NETWORK
TITLE = S006::STEP 006:TRAN 007: Pressure below setpoint?
//----------------------------------------------------------------------------//
// TRAN   TRAN   TRAN   TRAN   TRAN   TRAN   TRAN   TRAN   TRAN   TRAN   TRAN //
// TRAN   TRAN   TRAN   TRAN   TRAN   TRAN   TRAN   TRAN   TRAN   TRAN   TRAN //
//----------------------------------------------------------------------------//
// Pressure reduced below PRES_VAC.
//----------------------------------------------------------------------------//
// CONDITION   CONDITION   CONDITION   CONDITION   CONDITION   CONDITION   CO //
// CONDITION   CONDITION   CONDITION   CONDITION   CONDITION   CONDITION   CO //
//----------------------------------------------------------------------------//
      A(;
      L #_emc_gas_pi_vessel_pv;
      L #_r_pres_vac;
      <R;
      );






  //============================= TRAN FOOTER ==============================//
  // Transition jump control:                                               //
  //------------------------------------------------------------------------//
      A #sqSequencer.STEP.JumpCtrl;
      S #sqSequencer.STEP.Jump;
      S #sqSequencer.STEP.jumpDone[06];

NETWORK
TITLE = S006:t007::TRANS-v: EXIT TRANSITION AND READY THE NEXT STEP
//------------------------------------------------------------------------//
// Check the jump flag and jump to the next step if the transition        //
// condition is true and has set the jump flag:                           //
//------------------------------------------------------------------------//
      A #sqSequencer.STEP.Jump;
      JCN x007;

      R #sqSequencer.STEP.Jump;
      R #sqSequencer.STEP.Finished;

      L 08   ;// Load next STEPNO to jump to if transition satisfied
      T #sqSequencer.STEP.NumberNext;//Next Step08.

      JU COMM            ;// Transition satisfied, Exit, go to next step
x007:      NOP 0;






NETWORK
TITLE = S006::STEP-006:EXIT TRANSITION:
//========================== STEP TRANSFER ===============================//
// Jump to the common step progression code:                              //
//------------------------------------------------------------------------//
      JU COMM;






NETWORK
TITLE = S007: STEP-07::UO_MX_SETUP : Vacuum hold evacuation failed
//================================ STEP HEADER ===========================//
// STEP007 STEP007 STEP007 STEP007
// AUTOCODE   AUTOCODE   AUTOCODE   AUTOCODE   AUTOCODE   AUTOCODE   AUTO //
// STEP007 STEP007 STEP007 STEP007
//------------------------------------------------------------------------//
// Raise vacuum failed message.
// Log vacuum ejector time failed.
// Prompt operator to confirm to try again.
//------------------------------------------------------------------------//
S007:      NOP 0;

      SET;
      R #sqSequencer.STEP.jumpDone[07];
      A #sqSequencer.CMD.Pause;//If paused jump
      JC COMM;

NETWORK
TITLE = S007:STEP-07:Begin Action

      A #sqSequencer.STEP.Finished;
      JC A007;// Exit Action code, Jump to A007 Transition code

    //----------------------------------------------------------------------//
    // Begin step Action:                                                   //
    //----------------------------------------------------------------------//
      A #sqSequencer.STEP.Active;
      JC L007;// Action number loaded, Jump to L007--Step Action List

    //----------------------------------------------------------------------//
    // Load Default/Initial Step action number:                             //
    //----------------------------------------------------------------------//
      S #sqSequencer.STEP.Active;
      S #sqStepTimer.IN;
      L 1;//First Action, Step must contain Minimum one action
      T #sqSequencer.STEP.ActionNumber;

//----------------------------------------------------------------------------//
// Step action list.                                                          //
// aann=mini Action step number(aa) inside main step number(nn)               //
// First Action aa00, Second action ab00, Third ac00, etc.                    //
//----------------------------------------------------------------------------//
L007:      NOP 0;

      L #sqSequencer.STEP.ActionNumber;
      JL r007;//Wrong Action number
      JU _007;//Action error handling
      JU aa07;//ACTION-01


//----------------------------------------------------------------------------//
// More step action in the list can be inserted here, upto ab is tested:      //
//----------------------------------------------------------------------------//
r007:      NOP 0;//Wrong action number
      S #sqSequencer.Error_Fault;
      JU k007;//Exit
_007:      NOP 0;// Action error handling
      JU k007;// Exit






NETWORK
TITLE = S007:: STEP-007:: : ACTION CODE
//================================ ACT HEADER ============================//
// ACTION ACTION ACTION ACTION ACTION ACTION ACTION ACTION ACTION ACTION  //
// AUTOCODE   AUTOCODE   AUTOCODE   AUTOCODE   AUTOCODE   AUTOCODE   AUTO //
// ACTION ACTION ACTION ACTION ACTION ACTION ACTION ACTION ACTION ACTION  //
//------------------------------------------------------------------------//
// //Raise vacuum failed message.
// //Log vacuum time failed.
// //Prompt operator to confirm to try again.
aa07:      NOP 0;

  //------------------------------------------------------------------------//
  // ACT ACT ACT ACT ACT ACT ACT ACT ACT ACT ACT ACT ACT ACT ACT ACT ACT    //
  //------------------------------------------------------------------------//
  //Set flag to raise vacuum failed message
      SET;
      S #_log_real_vacuum_fail;
      S #_prompt_not_reach;

//Log pressure after vacuum timer expired(TIME_EJECT failed).
      L #_emc_gas_pi_vessel_pv;
      T #_real_vacuum_fail;

  //------------------------------------------------------------------------//
  // VERIFY  VERIFY VERIFY VERIFY VERIFY VERIFY VERIFY VERIFY VERIFY VERIFY //
  //------------------------------------------------------------------------//
      A "uncondJump";
      S #sqSequencer.STEP.ActionVerified;//Action verified

  //------------------------------------------------------------------------//
  // Action done:                                                           //
  //------------------------------------------------------------------------//
      O #sqSequencer.STEP.ActionVerified;
      O #smc.NO_VERIFIC     ;//No verification , bypass verification code
      S #sqSequencer.STEP.ActionFinished;






  //============================= STEP FOOTER ==============================//
  // AUTOCODE   AUTOCODE   AUTOCODE   AUTOCODE   AUTOCODE   AUTOCODE   AUTO //
  // Get Ready after action finished:                                       //
  //------------------------------------------------------------------------//
      A #sqSequencer.STEP.ActionFinished;
      JCN k007;

  //------------------------------------------------------------------------//
  // Reset Action finished flag, ready for next step action:                //
  //------------------------------------------------------------------------//
      R #sqSequencer.STEP.ActionVerified;
      R #sqSequencer.STEP.ActionFinished;

  //------------------------------------------------------------------------//
  // If ALL actions are finished:                                           //
  //------------------------------------------------------------------------//
      SET;
      S #sqSequencer.STEP.Finished;
      R #sqSequencer.STEP.Active;
      S #sqSequencer.STEP.Done[07];

  //------------------------------------------------------------------------//
  // End Step action(s):                                                    //
  //------------------------------------------------------------------------//
      JU k007;

//----------------------------------------------------------------------------//
// Finished Step Action(s):                                                   //
//----------------------------------------------------------------------------//
k007:      NOP 0;

      A #sqStepTimerExpired;
      S #sqSequencer.STEP.WithError[07];// Step error flag
      S #sqSequencer.Error_Fault;
      R #sqStepTimer.IN;

NETWORK
TITLE = S007:STEP-007::Begin Transition
//------------------------------------------------------------------------//
// Begin the transition code:                                             //
//------------------------------------------------------------------------//
A007:      NOP 0;
      R #sqStepTimer.IN;






  //============================= TRAN HEADER ==============================//
  // AUTOCODE   AUTOCODE   AUTOCODE   AUTOCODE   AUTOCODE   AUTOCODE   AUTO //
  // Bypass transition if manual jump:                                      //
  //------------------------------------------------------------------------//
      A #sqSequencer.STEP.Finished;
      A #smc.TRN_AND_JUMP   ;//Manual jump is set Transition as bypassed
      JCN COMM            ;//exit

NETWORK
TITLE = S007::STEP 007:TRAN 008: Try again?
//----------------------------------------------------------------------------//
// TRAN   TRAN   TRAN   TRAN   TRAN   TRAN   TRAN   TRAN   TRAN   TRAN   TRAN //
// TRAN   TRAN   TRAN   TRAN   TRAN   TRAN   TRAN   TRAN   TRAN   TRAN   TRAN //
//----------------------------------------------------------------------------//
// Operator want to try again.
//----------------------------------------------------------------------------//
// CONDITION   CONDITION   CONDITION   CONDITION   CONDITION   CONDITION   CO //
// CONDITION   CONDITION   CONDITION   CONDITION   CONDITION   CONDITION   CO //
//----------------------------------------------------------------------------//
      A #_prompt_not_reach_confirm_yes;






  //============================= TRAN FOOTER ==============================//
  // Transition jump control:                                               //
  //------------------------------------------------------------------------//
      A #sqSequencer.STEP.JumpCtrl;
      S #sqSequencer.STEP.Jump;
      S #sqSequencer.STEP.jumpDone[07];

NETWORK
TITLE = S007:t008::TRANS-v: EXIT TRANSITION AND READY THE NEXT STEP
//------------------------------------------------------------------------//
// Check the jump flag and jump to the next step if the transition        //
// condition is true and has set the jump flag:                           //
//------------------------------------------------------------------------//
      A #sqSequencer.STEP.Jump;
      JCN x008;

      R #sqSequencer.STEP.Jump;
      R #sqSequencer.STEP.Finished;

      L 09   ;// Load next STEPNO to jump to if transition satisfied
      T #sqSequencer.STEP.NumberNext;//Next Step09.

      JU COMM            ;// Transition satisfied, Exit, go to next step
x008:      NOP 0;






  //============================= TRAN HEADER ==============================//
  // AUTOCODE   AUTOCODE   AUTOCODE   AUTOCODE   AUTOCODE   AUTOCODE   AUTO //
  // Bypass transition if manual jump:                                      //
  //------------------------------------------------------------------------//
      A #sqSequencer.STEP.Finished;
      A #smc.TRN_AND_JUMP   ;//Manual jump is set Transition as bypassed
      JCN COMM            ;//exit

NETWORK
TITLE = S007::STEP 007:TRAN 009: No try?
//----------------------------------------------------------------------------//
// TRAN   TRAN   TRAN   TRAN   TRAN   TRAN   TRAN   TRAN   TRAN   TRAN   TRAN //
// TRAN   TRAN   TRAN   TRAN   TRAN   TRAN   TRAN   TRAN   TRAN   TRAN   TRAN //
//----------------------------------------------------------------------------//
// Operator don't want to try again.
//----------------------------------------------------------------------------//
// CONDITION   CONDITION   CONDITION   CONDITION   CONDITION   CONDITION   CO //
// CONDITION   CONDITION   CONDITION   CONDITION   CONDITION   CONDITION   CO //
//----------------------------------------------------------------------------//
      A #_prompt_not_reach_confirm_no;






  //============================= TRAN FOOTER ==============================//
  // Transition jump control:                                               //
  //------------------------------------------------------------------------//
      A #sqSequencer.STEP.JumpCtrl;
      S #sqSequencer.STEP.Jump;
      S #sqSequencer.STEP.jumpDone[07];

NETWORK
TITLE = S007:t009::TRANS-v: EXIT TRANSITION AND READY THE NEXT STEP
//------------------------------------------------------------------------//
// Check the jump flag and jump to the next step if the transition        //
// condition is true and has set the jump flag:                           //
//------------------------------------------------------------------------//
      A #sqSequencer.STEP.Jump;
      JCN x009;

      R #sqSequencer.STEP.Jump;
      R #sqSequencer.STEP.Finished;

      L 10   ;// Load next STEPNO to jump to if transition satisfied
      T #sqSequencer.STEP.NumberNext;//Next Step10.

      JU COMM            ;// Transition satisfied, Exit, go to next step
x009:      NOP 0;






NETWORK
TITLE = S007::STEP-007:EXIT TRANSITION:
//========================== STEP TRANSFER ===============================//
// Jump to the common step progression code:                              //
//------------------------------------------------------------------------//
      JU COMM;






NETWORK
TITLE = S008: STEP-08::UO_MX_SETUP : Start Vacuum Hold Timer
//================================ STEP HEADER ===========================//
// STEP008 STEP008 STEP008 STEP008
// AUTOCODE   AUTOCODE   AUTOCODE   AUTOCODE   AUTOCODE   AUTOCODE   AUTO //
// STEP008 STEP008 STEP008 STEP008
//------------------------------------------------------------------------//
// Close Mx vent line vacuum valve.
// Start Vacuum  Hold Timer.
// Store Vacuum Hold test begin time.
//------------------------------------------------------------------------//
S008:      NOP 0;

      SET;
      R #sqSequencer.STEP.jumpDone[08];
      A #sqSequencer.CMD.Pause;//If paused jump
      JC COMM;

NETWORK
TITLE = S008:STEP-08:Begin Action

      A #sqSequencer.STEP.Finished;
      JC A008;// Exit Action code, Jump to A008 Transition code

    //----------------------------------------------------------------------//
    // Begin step Action:                                                   //
    //----------------------------------------------------------------------//
      A #sqSequencer.STEP.Active;
      JC L008;// Action number loaded, Jump to L008--Step Action List

    //----------------------------------------------------------------------//
    // Load Default/Initial Step action number:                             //
    //----------------------------------------------------------------------//
      S #sqSequencer.STEP.Active;
      S #sqStepTimer.IN;
      L 1;//First Action, Step must contain Minimum one action
      T #sqSequencer.STEP.ActionNumber;

//----------------------------------------------------------------------------//
// Step action list.                                                          //
// aann=mini Action step number(aa) inside main step number(nn)               //
// First Action aa00, Second action ab00, Third ac00, etc.                    //
//----------------------------------------------------------------------------//
L008:      NOP 0;

      L #sqSequencer.STEP.ActionNumber;
      JL r008;//Wrong Action number
      JU _008;//Action error handling
      JU aa08;//ACTION-01
      JU ab08;//ACTION-02


//----------------------------------------------------------------------------//
// More step action in the list can be inserted here, upto ab is tested:      //
//----------------------------------------------------------------------------//
r008:      NOP 0;//Wrong action number
      S #sqSequencer.Error_Fault;
      JU k008;//Exit
_008:      NOP 0;// Action error handling
      JU k008;// Exit






NETWORK
TITLE = S008:: STEP-008:: : ACTION CODE
//================================ ACT HEADER ============================//
// ACTION ACTION ACTION ACTION ACTION ACTION ACTION ACTION ACTION ACTION  //
// AUTOCODE   AUTOCODE   AUTOCODE   AUTOCODE   AUTOCODE   AUTOCODE   AUTO //
// ACTION ACTION ACTION ACTION ACTION ACTION ACTION ACTION ACTION ACTION  //
//------------------------------------------------------------------------//
// //Close Mx vacuum valves.
aa08:      NOP 0;

  //------------------------------------------------------------------------//
  // ACT ACT ACT ACT ACT ACT ACT ACT ACT ACT ACT ACT ACT ACT ACT ACT ACT    //
  //------------------------------------------------------------------------//
  //Close Mx vacuum valve.
      L "dbCONST".SEL.GAS.NONE;
      T #_emc_gas_medium_gas;
      L "dbCONST".BLK.CMD.RESTART;
      T #_emc_gas_cmd;

// Reset vacuum hold timer
      R #sqSeqTimerStart;

  //------------------------------------------------------------------------//
  // VERIFY  VERIFY VERIFY VERIFY VERIFY VERIFY VERIFY VERIFY VERIFY VERIFY //
  //------------------------------------------------------------------------//
      AN #SQ_TIMER.Q;
      A(;
      L #_emc_gas_state;
      L "dbCONST".BLK.STATE.STOPPED;
      >I;
      );
      A(;
      L #_emc_gas_state;
      L "dbCONST".BLK.STATE.INTERLOCKED;
      <I;
      );
      S #sqSequencer.STEP.ActionVerified;//Action verified

  //------------------------------------------------------------------------//
  // Action done:                                                           //
  //------------------------------------------------------------------------//
      O #sqSequencer.STEP.ActionVerified;
      O #smc.NO_VERIFIC     ;//No verification , bypass verification code
      S #sqSequencer.STEP.ActionFinished;






  //============================= ACT FOOTER ===============================//
  // AUTOCODE   AUTOCODE   AUTOCODE   AUTOCODE   AUTOCODE   AUTOCODE   AUTO //
  // Get Ready after action finished:                                       //
  //------------------------------------------------------------------------//
      A #sqSequencer.STEP.ActionFinished;
      JCN k008;

  //------------------------------------------------------------------------//
  // Reset Action finished flag, ready for next step action:                //
  //------------------------------------------------------------------------//
      R #sqSequencer.STEP.ActionVerified;
      R #sqSequencer.STEP.ActionFinished;

  //------------------------------------------------------------------------//
  // Load Next Step Action number:                                          //
  //------------------------------------------------------------------------//
      L 02;//Load next Action
      T #sqSequencer.STEP.ActionNumber;






NETWORK
TITLE = S008:: STEP-008:: : ACTION CODE
//================================ ACT HEADER ============================//
// ACTION ACTION ACTION ACTION ACTION ACTION ACTION ACTION ACTION ACTION  //
// AUTOCODE   AUTOCODE   AUTOCODE   AUTOCODE   AUTOCODE   AUTOCODE   AUTO //
// ACTION ACTION ACTION ACTION ACTION ACTION ACTION ACTION ACTION ACTION  //
//------------------------------------------------------------------------//
// //Start Vacuum Hold Timer.
// //Store Vacuum Hold test begin time.
ab08:      NOP 0;

  //------------------------------------------------------------------------//
  // ACT ACT ACT ACT ACT ACT ACT ACT ACT ACT ACT ACT ACT ACT ACT ACT ACT    //
  //------------------------------------------------------------------------//
      L "dbCONST".BLK.CMD.START;
      T #_emc_gas_cmd;

// Start vacuum hold timer
      L #_r_time_vac_hold;
      T #SQ_TIMER.PT;
      S #sqSeqTimerStart;

//Store Vacuum Hold test begin time.
      L "dbCONST".CHRONO.CPU_TIME;
      T #_vacuum_held_begin_time;

  //------------------------------------------------------------------------//
  // VERIFY  VERIFY VERIFY VERIFY VERIFY VERIFY VERIFY VERIFY VERIFY VERIFY //
  //------------------------------------------------------------------------//
      A #sqSeqTimerStart;
      S #sqSequencer.STEP.ActionVerified;//Action verified

  //------------------------------------------------------------------------//
  // Action done:                                                           //
  //------------------------------------------------------------------------//
      O #sqSequencer.STEP.ActionVerified;
      O #smc.NO_VERIFIC     ;//No verification , bypass verification code
      S #sqSequencer.STEP.ActionFinished;






  //============================= STEP FOOTER ==============================//
  // AUTOCODE   AUTOCODE   AUTOCODE   AUTOCODE   AUTOCODE   AUTOCODE   AUTO //
  // Get Ready after action finished:                                       //
  //------------------------------------------------------------------------//
      A #sqSequencer.STEP.ActionFinished;
      JCN k008;

  //------------------------------------------------------------------------//
  // Reset Action finished flag, ready for next step action:                //
  //------------------------------------------------------------------------//
      R #sqSequencer.STEP.ActionVerified;
      R #sqSequencer.STEP.ActionFinished;

  //------------------------------------------------------------------------//
  // If ALL actions are finished:                                           //
  //------------------------------------------------------------------------//
      SET;
      S #sqSequencer.STEP.Finished;
      R #sqSequencer.STEP.Active;
      S #sqSequencer.STEP.Done[08];

  //------------------------------------------------------------------------//
  // End Step action(s):                                                    //
  //------------------------------------------------------------------------//
      JU k008;

//----------------------------------------------------------------------------//
// Finished Step Action(s):                                                   //
//----------------------------------------------------------------------------//
k008:      NOP 0;

      A #sqStepTimerExpired;
      S #sqSequencer.STEP.WithError[08];// Step error flag
      S #sqSequencer.Error_Fault;
      R #sqStepTimer.IN;

NETWORK
TITLE = S008:STEP-008::Begin Transition
//------------------------------------------------------------------------//
// Begin the transition code:                                             //
//------------------------------------------------------------------------//
A008:      NOP 0;
      R #sqStepTimer.IN;






  //============================= TRAN HEADER ==============================//
  // AUTOCODE   AUTOCODE   AUTOCODE   AUTOCODE   AUTOCODE   AUTOCODE   AUTO //
  // Bypass transition if manual jump:                                      //
  //------------------------------------------------------------------------//
      A #sqSequencer.STEP.Finished;
      A #smc.TRN_AND_JUMP   ;//Manual jump is set Transition as bypassed
      JCN COMM            ;//exit

NETWORK
TITLE = S008::STEP 008:TRAN 010: Jump when gas command completed
//----------------------------------------------------------------------------//
// TRAN   TRAN   TRAN   TRAN   TRAN   TRAN   TRAN   TRAN   TRAN   TRAN   TRAN //
// TRAN   TRAN   TRAN   TRAN   TRAN   TRAN   TRAN   TRAN   TRAN   TRAN   TRAN //
//----------------------------------------------------------------------------//
//
//----------------------------------------------------------------------------//
// CONDITION   CONDITION   CONDITION   CONDITION   CONDITION   CONDITION   CO //
// CONDITION   CONDITION   CONDITION   CONDITION   CONDITION   CONDITION   CO //
//----------------------------------------------------------------------------//
      A(;
      L #_emc_gas_state;
      L "dbCONST".BLK.STATE.COMPLETED;
      ==I;
      );






  //============================= TRAN FOOTER ==============================//
  // Transition jump control:                                               //
  //------------------------------------------------------------------------//
      A #sqSequencer.STEP.JumpCtrl;
      S #sqSequencer.STEP.Jump;
      S #sqSequencer.STEP.jumpDone[08];

NETWORK
TITLE = S008:t010::TRANS-v: EXIT TRANSITION AND READY THE NEXT STEP
//------------------------------------------------------------------------//
// Check the jump flag and jump to the next step if the transition        //
// condition is true and has set the jump flag:                           //
//------------------------------------------------------------------------//
      A #sqSequencer.STEP.Jump;
      JCN x010;

      R #sqSequencer.STEP.Jump;
      R #sqSequencer.STEP.Finished;

      L 11   ;// Load next STEPNO to jump to if transition satisfied
      T #sqSequencer.STEP.NumberNext;//Next Step11.

      JU COMM            ;// Transition satisfied, Exit, go to next step
x010:      NOP 0;






NETWORK
TITLE = S008::STEP-008:EXIT TRANSITION:
//========================== STEP TRANSFER ===============================//
// Jump to the common step progression code:                              //
//------------------------------------------------------------------------//
      JU COMM;






NETWORK
TITLE = S009: STEP-09::UO_MX_SETUP : Log operator repeat
//================================ STEP HEADER ===========================//
// STEP009 STEP009 STEP009 STEP009
// AUTOCODE   AUTOCODE   AUTOCODE   AUTOCODE   AUTOCODE   AUTOCODE   AUTO //
// STEP009 STEP009 STEP009 STEP009
//------------------------------------------------------------------------//
// Log operator repeat.
//------------------------------------------------------------------------//
S009:      NOP 0;

      SET;
      R #sqSequencer.STEP.jumpDone[09];
      A #sqSequencer.CMD.Pause;//If paused jump
      JC COMM;

NETWORK
TITLE = S009:STEP-09:Begin Action

      A #sqSequencer.STEP.Finished;
      JC A009;// Exit Action code, Jump to A009 Transition code

    //----------------------------------------------------------------------//
    // Begin step Action:                                                   //
    //----------------------------------------------------------------------//
      A #sqSequencer.STEP.Active;
      JC L009;// Action number loaded, Jump to L009--Step Action List

    //----------------------------------------------------------------------//
    // Load Default/Initial Step action number:                             //
    //----------------------------------------------------------------------//
      S #sqSequencer.STEP.Active;
      S #sqStepTimer.IN;
      L 1;//First Action, Step must contain Minimum one action
      T #sqSequencer.STEP.ActionNumber;

//----------------------------------------------------------------------------//
// Step action list.                                                          //
// aann=mini Action step number(aa) inside main step number(nn)               //
// First Action aa00, Second action ab00, Third ac00, etc.                    //
//----------------------------------------------------------------------------//
L009:      NOP 0;

      L #sqSequencer.STEP.ActionNumber;
      JL r009;//Wrong Action number
      JU _009;//Action error handling
      JU aa09;//ACTION-01


//----------------------------------------------------------------------------//
// More step action in the list can be inserted here, upto ab is tested:      //
//----------------------------------------------------------------------------//
r009:      NOP 0;//Wrong action number
      S #sqSequencer.Error_Fault;
      JU k009;//Exit
_009:      NOP 0;// Action error handling
      JU k009;// Exit






NETWORK
TITLE = S009:: STEP-009:: : ACTION CODE
//================================ ACT HEADER ============================//
// ACTION ACTION ACTION ACTION ACTION ACTION ACTION ACTION ACTION ACTION  //
// AUTOCODE   AUTOCODE   AUTOCODE   AUTOCODE   AUTOCODE   AUTOCODE   AUTO //
// ACTION ACTION ACTION ACTION ACTION ACTION ACTION ACTION ACTION ACTION  //
//------------------------------------------------------------------------//
// //Log operator repeat.
aa09:      NOP 0;

  //------------------------------------------------------------------------//
  // ACT ACT ACT ACT ACT ACT ACT ACT ACT ACT ACT ACT ACT ACT ACT ACT ACT    //
  //------------------------------------------------------------------------//
  //Log operator repeat.
      SET;
      S #_log_msg_not_reach_repeat;
      R #_prompt_not_reach_confirm_yes;
      R #sqSeqTimerStart;

  //------------------------------------------------------------------------//
  // VERIFY  VERIFY VERIFY VERIFY VERIFY VERIFY VERIFY VERIFY VERIFY VERIFY //
  //------------------------------------------------------------------------//
      A "uncondJump";
      S #sqSequencer.STEP.ActionVerified;//Action verified

  //------------------------------------------------------------------------//
  // Action done:                                                           //
  //------------------------------------------------------------------------//
      O #sqSequencer.STEP.ActionVerified;
      O #smc.NO_VERIFIC     ;//No verification , bypass verification code
      S #sqSequencer.STEP.ActionFinished;






  //============================= STEP FOOTER ==============================//
  // AUTOCODE   AUTOCODE   AUTOCODE   AUTOCODE   AUTOCODE   AUTOCODE   AUTO //
  // Get Ready after action finished:                                       //
  //------------------------------------------------------------------------//
      A #sqSequencer.STEP.ActionFinished;
      JCN k009;

  //------------------------------------------------------------------------//
  // Reset Action finished flag, ready for next step action:                //
  //------------------------------------------------------------------------//
      R #sqSequencer.STEP.ActionVerified;
      R #sqSequencer.STEP.ActionFinished;

  //------------------------------------------------------------------------//
  // If ALL actions are finished:                                           //
  //------------------------------------------------------------------------//
      SET;
      S #sqSequencer.STEP.Finished;
      R #sqSequencer.STEP.Active;
      S #sqSequencer.STEP.Done[09];

  //------------------------------------------------------------------------//
  // End Step action(s):                                                    //
  //------------------------------------------------------------------------//
      JU k009;

//----------------------------------------------------------------------------//
// Finished Step Action(s):                                                   //
//----------------------------------------------------------------------------//
k009:      NOP 0;

      A #sqStepTimerExpired;
      S #sqSequencer.STEP.WithError[09];// Step error flag
      S #sqSequencer.Error_Fault;
      R #sqStepTimer.IN;

NETWORK
TITLE = S009:STEP-009::Begin Transition
//------------------------------------------------------------------------//
// Begin the transition code:                                             //
//------------------------------------------------------------------------//
A009:      NOP 0;
      R #sqStepTimer.IN;






  //============================= TRAN HEADER ==============================//
  // AUTOCODE   AUTOCODE   AUTOCODE   AUTOCODE   AUTOCODE   AUTOCODE   AUTO //
  // Bypass transition if manual jump:                                      //
  //------------------------------------------------------------------------//
      A #sqSequencer.STEP.Finished;
      A #smc.TRN_AND_JUMP   ;//Manual jump is set Transition as bypassed
      JCN COMM            ;//exit

NETWORK
TITLE = S009::STEP 009:TRAN 011: Empty Transition
//----------------------------------------------------------------------------//
// TRAN   TRAN   TRAN   TRAN   TRAN   TRAN   TRAN   TRAN   TRAN   TRAN   TRAN //
// TRAN   TRAN   TRAN   TRAN   TRAN   TRAN   TRAN   TRAN   TRAN   TRAN   TRAN //
//----------------------------------------------------------------------------//
// Empty Transition
//----------------------------------------------------------------------------//
// CONDITION   CONDITION   CONDITION   CONDITION   CONDITION   CONDITION   CO //
// CONDITION   CONDITION   CONDITION   CONDITION   CONDITION   CONDITION   CO //
//----------------------------------------------------------------------------//
      A "uncondJump";






  //============================= TRAN FOOTER ==============================//
  // Transition jump control:                                               //
  //------------------------------------------------------------------------//
      A #sqSequencer.STEP.JumpCtrl;
      S #sqSequencer.STEP.Jump;
      S #sqSequencer.STEP.jumpDone[09];

NETWORK
TITLE = S009:t011::TRANS-v: EXIT TRANSITION AND READY THE NEXT STEP
//------------------------------------------------------------------------//
// Check the jump flag and jump to the next step if the transition        //
// condition is true and has set the jump flag:                           //
//------------------------------------------------------------------------//
      A #sqSequencer.STEP.Jump;
      JCN x011;

      R #sqSequencer.STEP.Jump;
      R #sqSequencer.STEP.Finished;

      L 06   ;// Load next STEPNO to jump to if transition satisfied
      T #sqSequencer.STEP.NumberNext;//Next Step06.

      JU COMM            ;// Transition satisfied, Exit, go to next step
x011:      NOP 0;






NETWORK
TITLE = S009::STEP-009:EXIT TRANSITION:
//========================== STEP TRANSFER ===============================//
// Jump to the common step progression code:                              //
//------------------------------------------------------------------------//
      JU COMM;






NETWORK
TITLE = S010: STEP-10::UO_MX_SETUP : Log operator abort
//================================ STEP HEADER ===========================//
// STEP010 STEP010 STEP010 STEP010
// AUTOCODE   AUTOCODE   AUTOCODE   AUTOCODE   AUTOCODE   AUTOCODE   AUTO //
// STEP010 STEP010 STEP010 STEP010
//------------------------------------------------------------------------//
// Log operator abort.
//------------------------------------------------------------------------//
S010:      NOP 0;

      SET;
      R #sqSequencer.STEP.jumpDone[10];
      A #sqSequencer.CMD.Pause;//If paused jump
      JC COMM;

NETWORK
TITLE = S010:STEP-10:Begin Action

      A #sqSequencer.STEP.Finished;
      JC A010;// Exit Action code, Jump to A010 Transition code

    //----------------------------------------------------------------------//
    // Begin step Action:                                                   //
    //----------------------------------------------------------------------//
      A #sqSequencer.STEP.Active;
      JC L010;// Action number loaded, Jump to L010--Step Action List

    //----------------------------------------------------------------------//
    // Load Default/Initial Step action number:                             //
    //----------------------------------------------------------------------//
      S #sqSequencer.STEP.Active;
      S #sqStepTimer.IN;
      L 1;//First Action, Step must contain Minimum one action
      T #sqSequencer.STEP.ActionNumber;

//----------------------------------------------------------------------------//
// Step action list.                                                          //
// aann=mini Action step number(aa) inside main step number(nn)               //
// First Action aa00, Second action ab00, Third ac00, etc.                    //
//----------------------------------------------------------------------------//
L010:      NOP 0;

      L #sqSequencer.STEP.ActionNumber;
      JL r010;//Wrong Action number
      JU _010;//Action error handling
      JU aa10;//ACTION-01


//----------------------------------------------------------------------------//
// More step action in the list can be inserted here, upto ab is tested:      //
//----------------------------------------------------------------------------//
r010:      NOP 0;//Wrong action number
      S #sqSequencer.Error_Fault;
      JU k010;//Exit
_010:      NOP 0;// Action error handling
      JU k010;// Exit






NETWORK
TITLE = S010:: STEP-010:: : ACTION CODE
//================================ ACT HEADER ============================//
// ACTION ACTION ACTION ACTION ACTION ACTION ACTION ACTION ACTION ACTION  //
// AUTOCODE   AUTOCODE   AUTOCODE   AUTOCODE   AUTOCODE   AUTOCODE   AUTO //
// ACTION ACTION ACTION ACTION ACTION ACTION ACTION ACTION ACTION ACTION  //
//------------------------------------------------------------------------//
// //Log operator ABORT.
aa10:      NOP 0;

  //------------------------------------------------------------------------//
  // ACT ACT ACT ACT ACT ACT ACT ACT ACT ACT ACT ACT ACT ACT ACT ACT ACT    //
  //------------------------------------------------------------------------//
  //Log operator abort.
      SET;
      S #_log_msg_not_reach_abort;
      R #_prompt_not_reach_confirm_no;
      R #sqSeqTimerStart;

  //------------------------------------------------------------------------//
  // VERIFY  VERIFY VERIFY VERIFY VERIFY VERIFY VERIFY VERIFY VERIFY VERIFY //
  //------------------------------------------------------------------------//
      A "uncondJump";
      S #sqSequencer.STEP.ActionVerified;//Action verified

  //------------------------------------------------------------------------//
  // Action done:                                                           //
  //------------------------------------------------------------------------//
      O #sqSequencer.STEP.ActionVerified;
      O #smc.NO_VERIFIC     ;//No verification , bypass verification code
      S #sqSequencer.STEP.ActionFinished;






  //============================= STEP FOOTER ==============================//
  // AUTOCODE   AUTOCODE   AUTOCODE   AUTOCODE   AUTOCODE   AUTOCODE   AUTO //
  // Get Ready after action finished:                                       //
  //------------------------------------------------------------------------//
      A #sqSequencer.STEP.ActionFinished;
      JCN k010;

  //------------------------------------------------------------------------//
  // Reset Action finished flag, ready for next step action:                //
  //------------------------------------------------------------------------//
      R #sqSequencer.STEP.ActionVerified;
      R #sqSequencer.STEP.ActionFinished;

  //------------------------------------------------------------------------//
  // If ALL actions are finished:                                           //
  //------------------------------------------------------------------------//
      SET;
      S #sqSequencer.STEP.Finished;
      R #sqSequencer.STEP.Active;
      S #sqSequencer.STEP.Done[10];

  //------------------------------------------------------------------------//
  // End Step action(s):                                                    //
  //------------------------------------------------------------------------//
      JU k010;

//----------------------------------------------------------------------------//
// Finished Step Action(s):                                                   //
//----------------------------------------------------------------------------//
k010:      NOP 0;

      A #sqStepTimerExpired;
      S #sqSequencer.STEP.WithError[10];// Step error flag
      S #sqSequencer.Error_Fault;
      R #sqStepTimer.IN;

NETWORK
TITLE = S010:STEP-010::Begin Transition
//------------------------------------------------------------------------//
// Begin the transition code:                                             //
//------------------------------------------------------------------------//
A010:      NOP 0;
      R #sqStepTimer.IN;






  //============================= TRAN HEADER ==============================//
  // AUTOCODE   AUTOCODE   AUTOCODE   AUTOCODE   AUTOCODE   AUTOCODE   AUTO //
  // Bypass transition if manual jump:                                      //
  //------------------------------------------------------------------------//
      A #sqSequencer.STEP.Finished;
      A #smc.TRN_AND_JUMP   ;//Manual jump is set Transition as bypassed
      JCN COMM            ;//exit

NETWORK
TITLE = S010::STEP 010:TRAN 012: Empty Transition
//----------------------------------------------------------------------------//
// TRAN   TRAN   TRAN   TRAN   TRAN   TRAN   TRAN   TRAN   TRAN   TRAN   TRAN //
// TRAN   TRAN   TRAN   TRAN   TRAN   TRAN   TRAN   TRAN   TRAN   TRAN   TRAN //
//----------------------------------------------------------------------------//
// Empty Transition
//----------------------------------------------------------------------------//
// CONDITION   CONDITION   CONDITION   CONDITION   CONDITION   CONDITION   CO //
// CONDITION   CONDITION   CONDITION   CONDITION   CONDITION   CONDITION   CO //
//----------------------------------------------------------------------------//
      A "uncondJump";






  //============================= TRAN FOOTER ==============================//
  // Transition jump control:                                               //
  //------------------------------------------------------------------------//
      A #sqSequencer.STEP.JumpCtrl;
      S #sqSequencer.STEP.Jump;
      S #sqSequencer.STEP.jumpDone[10];

NETWORK
TITLE = S010:t012::TRANS-v: EXIT TRANSITION AND READY THE NEXT STEP
//------------------------------------------------------------------------//
// Check the jump flag and jump to the next step if the transition        //
// condition is true and has set the jump flag:                           //
//------------------------------------------------------------------------//
      A #sqSequencer.STEP.Jump;
      JCN x012;

      R #sqSequencer.STEP.Jump;
      R #sqSequencer.STEP.Finished;

      L 17   ;// Load next STEPNO to jump to if transition satisfied
      T #sqSequencer.STEP.NumberNext;//Next Step17.

      JU COMM            ;// Transition satisfied, Exit, go to next step
x012:      NOP 0;






NETWORK
TITLE = S010::STEP-010:EXIT TRANSITION:
//========================== STEP TRANSFER ===============================//
// Jump to the common step progression code:                              //
//------------------------------------------------------------------------//
      JU COMM;






NETWORK
TITLE = S011: STEP-11::UO_MX_SETUP: Vacuum Hold Test
//================================ STEP HEADER ===========================//
// STEP011 STEP011 STEP011 STEP011
// AUTOCODE   AUTOCODE   AUTOCODE   AUTOCODE   AUTOCODE   AUTOCODE   AUTO //
// STEP011 STEP011 STEP011 STEP011
//------------------------------------------------------------------------//
//
//------------------------------------------------------------------------//
S011:      NOP 0;

      SET;
      R #sqSequencer.STEP.jumpDone[11];
      A #sqSequencer.CMD.Pause;//If paused jump
      JC COMM;

NETWORK
TITLE = S011:STEP-11:Begin Action

      A #sqSequencer.STEP.Finished;
      JC A011;// Exit Action code, Jump to A011 Transition code

    //----------------------------------------------------------------------//
    // Begin step Action:                                                   //
    //----------------------------------------------------------------------//
      A #sqSequencer.STEP.Active;
      JC L011;// Action number loaded, Jump to L011--Step Action List

    //----------------------------------------------------------------------//
    // Load Default/Initial Step action number:                             //
    //----------------------------------------------------------------------//
      S #sqSequencer.STEP.Active;
      S #sqStepTimer.IN;
      L 1;//First Action, Step must contain Minimum one action
      T #sqSequencer.STEP.ActionNumber;

//----------------------------------------------------------------------------//
// Step action list.                                                          //
// aann=mini Action step number(aa) inside main step number(nn)               //
// First Action aa00, Second action ab00, Third ac00, etc.                    //
//----------------------------------------------------------------------------//
L011:      NOP 0;

      L #sqSequencer.STEP.ActionNumber;
      JL r011;//Wrong Action number
      JU _011;//Action error handling
      JU aa11;//ACTION-01


//----------------------------------------------------------------------------//
// More step action in the list can be inserted here, upto ab is tested:      //
//----------------------------------------------------------------------------//
r011:      NOP 0;//Wrong action number
      S #sqSequencer.Error_Fault;
      JU k011;//Exit
_011:      NOP 0;// Action error handling
      JU k011;// Exit






NETWORK
TITLE = S011:: STEP-011:: : ACTION CODE
//================================ ACT HEADER ============================//
// ACTION ACTION ACTION ACTION ACTION ACTION ACTION ACTION ACTION ACTION  //
// AUTOCODE   AUTOCODE   AUTOCODE   AUTOCODE   AUTOCODE   AUTOCODE   AUTO //
// ACTION ACTION ACTION ACTION ACTION ACTION ACTION ACTION ACTION ACTION  //
//------------------------------------------------------------------------//
// //Clear gas EM restart command
aa11:      NOP 0;

  //------------------------------------------------------------------------//
  // ACT ACT ACT ACT ACT ACT ACT ACT ACT ACT ACT ACT ACT ACT ACT ACT ACT    //
  //------------------------------------------------------------------------//
      L "dbCONST".BLK.CMD.START;
      T #_emc_gas_cmd;

  //------------------------------------------------------------------------//
  // VERIFY  VERIFY VERIFY VERIFY VERIFY VERIFY VERIFY VERIFY VERIFY VERIFY //
  //------------------------------------------------------------------------//

      S #sqSequencer.STEP.ActionVerified;//Action verified

  //------------------------------------------------------------------------//
  // Action done:                                                           //
  //------------------------------------------------------------------------//
      O #sqSequencer.STEP.ActionVerified;
      O #smc.NO_VERIFIC     ;//No verification , bypass verification code
      S #sqSequencer.STEP.ActionFinished;






  //============================= STEP FOOTER ==============================//
  // AUTOCODE   AUTOCODE   AUTOCODE   AUTOCODE   AUTOCODE   AUTOCODE   AUTO //
  // Get Ready after action finished:                                       //
  //------------------------------------------------------------------------//
      A #sqSequencer.STEP.ActionFinished;
      JCN k011;

  //------------------------------------------------------------------------//
  // Reset Action finished flag, ready for next step action:                //
  //------------------------------------------------------------------------//
      R #sqSequencer.STEP.ActionVerified;
      R #sqSequencer.STEP.ActionFinished;

  //------------------------------------------------------------------------//
  // If ALL actions are finished:                                           //
  //------------------------------------------------------------------------//
      SET;
      S #sqSequencer.STEP.Finished;
      R #sqSequencer.STEP.Active;
      S #sqSequencer.STEP.Done[11];

  //------------------------------------------------------------------------//
  // End Step action(s):                                                    //
  //------------------------------------------------------------------------//
      JU k011;

//----------------------------------------------------------------------------//
// Finished Step Action(s):                                                   //
//----------------------------------------------------------------------------//
k011:      NOP 0;

      A #sqStepTimerExpired;
      S #sqSequencer.STEP.WithError[11];// Step error flag
      S #sqSequencer.Error_Fault;
      R #sqStepTimer.IN;

NETWORK
TITLE = S011:STEP-011::Begin Transition
//------------------------------------------------------------------------//
// Begin the transition code:                                             //
//------------------------------------------------------------------------//
A011:      NOP 0;
      R #sqStepTimer.IN;






  //============================= TRAN HEADER ==============================//
  // AUTOCODE   AUTOCODE   AUTOCODE   AUTOCODE   AUTOCODE   AUTOCODE   AUTO //
  // Bypass transition if manual jump:                                      //
  //------------------------------------------------------------------------//
      A #sqSequencer.STEP.Finished;
      A #smc.TRN_AND_JUMP   ;//Manual jump is set Transition as bypassed
      JCN COMM            ;//exit

NETWORK
TITLE = S011::STEP 011:TRAN 013: Empty Transition
//----------------------------------------------------------------------------//
// TRAN   TRAN   TRAN   TRAN   TRAN   TRAN   TRAN   TRAN   TRAN   TRAN   TRAN //
// TRAN   TRAN   TRAN   TRAN   TRAN   TRAN   TRAN   TRAN   TRAN   TRAN   TRAN //
//----------------------------------------------------------------------------//
// Empty Transition
//----------------------------------------------------------------------------//
// CONDITION   CONDITION   CONDITION   CONDITION   CONDITION   CONDITION   CO //
// CONDITION   CONDITION   CONDITION   CONDITION   CONDITION   CONDITION   CO //
//----------------------------------------------------------------------------//
      A "uncondJump";






  //============================= TRAN FOOTER ==============================//
  // Transition jump control:                                               //
  //------------------------------------------------------------------------//
      A #sqSequencer.STEP.JumpCtrl;
      S #sqSequencer.STEP.Jump;
      S #sqSequencer.STEP.jumpDone[11];

NETWORK
TITLE = S011:t013::TRANS-v: EXIT TRANSITION AND READY THE NEXT STEP
//------------------------------------------------------------------------//
// Check the jump flag and jump to the next step if the transition        //
// condition is true and has set the jump flag:                           //
//------------------------------------------------------------------------//
      A #sqSequencer.STEP.Jump;
      JCN x013;

      R #sqSequencer.STEP.Jump;
      R #sqSequencer.STEP.Finished;

      L 12   ;// Load next STEPNO to jump to if transition satisfied
      T #sqSequencer.STEP.NumberNext;//Next Step12.

      JU COMM            ;// Transition satisfied, Exit, go to next step
x013:      NOP 0;






NETWORK
TITLE = S011::STEP-011:EXIT TRANSITION:
//========================== STEP TRANSFER ===============================//
// Jump to the common step progression code:                              //
//------------------------------------------------------------------------//
      JU COMM;






NETWORK
TITLE = S012: STEP-12::UO_MX_SETUP : Pressure logging
//================================ STEP HEADER ===========================//
// STEP012 STEP012 STEP012 STEP012
// AUTOCODE   AUTOCODE   AUTOCODE   AUTOCODE   AUTOCODE   AUTOCODE   AUTO //
// STEP012 STEP012 STEP012 STEP012
//------------------------------------------------------------------------//
// Log vessel pressure at 30 second intervals.
//------------------------------------------------------------------------//
S012:      NOP 0;

      SET;
      R #sqSequencer.STEP.jumpDone[12];
      A #sqSequencer.CMD.Pause;//If paused jump
      JC COMM;

NETWORK
TITLE = S012:STEP-12:Begin Action

      A #sqSequencer.STEP.Finished;
      JC A012;// Exit Action code, Jump to A012 Transition code

    //----------------------------------------------------------------------//
    // Begin step Action:                                                   //
    //----------------------------------------------------------------------//
      A #sqSequencer.STEP.Active;
      JC L012;// Action number loaded, Jump to L012--Step Action List

    //----------------------------------------------------------------------//
    // Load Default/Initial Step action number:                             //
    //----------------------------------------------------------------------//
      S #sqSequencer.STEP.Active;
      S #sqStepTimer.IN;
      L 1;//First Action, Step must contain Minimum one action
      T #sqSequencer.STEP.ActionNumber;

//----------------------------------------------------------------------------//
// Step action list.                                                          //
// aann=mini Action step number(aa) inside main step number(nn)               //
// First Action aa00, Second action ab00, Third ac00, etc.                    //
//----------------------------------------------------------------------------//
L012:      NOP 0;

      L #sqSequencer.STEP.ActionNumber;
      JL r012;//Wrong Action number
      JU _012;//Action error handling
      JU aa12;//ACTION-01


//----------------------------------------------------------------------------//
// More step action in the list can be inserted here, upto ab is tested:      //
//----------------------------------------------------------------------------//
r012:      NOP 0;//Wrong action number
      S #sqSequencer.Error_Fault;
      JU k012;//Exit
_012:      NOP 0;// Action error handling
      JU k012;// Exit






NETWORK
TITLE = S012:: STEP-012:: : ACTION CODE
//================================ ACT HEADER ============================//
// ACTION ACTION ACTION ACTION ACTION ACTION ACTION ACTION ACTION ACTION  //
// AUTOCODE   AUTOCODE   AUTOCODE   AUTOCODE   AUTOCODE   AUTOCODE   AUTO //
// ACTION ACTION ACTION ACTION ACTION ACTION ACTION ACTION ACTION ACTION  //
//------------------------------------------------------------------------//
// //Set flags to log Sy vessel pressure.
aa12:      NOP 0;

  //------------------------------------------------------------------------//
  // ACT ACT ACT ACT ACT ACT ACT ACT ACT ACT ACT ACT ACT ACT ACT ACT ACT    //
  //------------------------------------------------------------------------//
  //Log Mx vessel pressure.
      L #_emc_gas_pi_vessel_pv;
      T #_real_pressure_mx;

      A #SQ_TIMER2.Q;
      R #sqSeqTimerStart2;
      R #_log_real_pressure_mx;

      AN #SQ_TIMER2.Q;
      S #sqSeqTimerStart2;
      S #_log_real_pressure_mx;
      L T#30S;
      T #SQ_TIMER2.PT;

  //------------------------------------------------------------------------//
  // VERIFY  VERIFY VERIFY VERIFY VERIFY VERIFY VERIFY VERIFY VERIFY VERIFY //
  //------------------------------------------------------------------------//
      A "uncondJump";
      S #sqSequencer.STEP.ActionVerified;//Action verified

  //------------------------------------------------------------------------//
  // Action done:                                                           //
  //------------------------------------------------------------------------//
      O #sqSequencer.STEP.ActionVerified;
      O #smc.NO_VERIFIC     ;//No verification , bypass verification code
      S #sqSequencer.STEP.ActionFinished;






  //============================= STEP FOOTER ==============================//
  // AUTOCODE   AUTOCODE   AUTOCODE   AUTOCODE   AUTOCODE   AUTOCODE   AUTO //
  // Get Ready after action finished:                                       //
  //------------------------------------------------------------------------//
      A #sqSequencer.STEP.ActionFinished;
      JCN k012;

  //------------------------------------------------------------------------//
  // Reset Action finished flag, ready for next step action:                //
  //------------------------------------------------------------------------//
      R #sqSequencer.STEP.ActionVerified;
      R #sqSequencer.STEP.ActionFinished;

  //------------------------------------------------------------------------//
  // If ALL actions are finished:                                           //
  //------------------------------------------------------------------------//
      SET;
      S #sqSequencer.STEP.Finished;
      R #sqSequencer.STEP.Active;
      S #sqSequencer.STEP.Done[12];

  //------------------------------------------------------------------------//
  // End Step action(s):                                                    //
  //------------------------------------------------------------------------//
      JU k012;

//----------------------------------------------------------------------------//
// Finished Step Action(s):                                                   //
//----------------------------------------------------------------------------//
k012:      NOP 0;

      A #sqStepTimerExpired;
      S #sqSequencer.STEP.WithError[12];// Step error flag
      S #sqSequencer.Error_Fault;
      R #sqStepTimer.IN;

NETWORK
TITLE = S012:STEP-012::Begin Transition
//------------------------------------------------------------------------//
// Begin the transition code:                                             //
//------------------------------------------------------------------------//
A012:      NOP 0;
      R #sqStepTimer.IN;






  //============================= TRAN HEADER ==============================//
  // AUTOCODE   AUTOCODE   AUTOCODE   AUTOCODE   AUTOCODE   AUTOCODE   AUTO //
  // Bypass transition if manual jump:                                      //
  //------------------------------------------------------------------------//
      A #sqSequencer.STEP.Finished;
      A #smc.TRN_AND_JUMP   ;//Manual jump is set Transition as bypassed
      JCN COMM            ;//exit

NETWORK
TITLE = S012::STEP 012:TRAN 014: Timer Expired
//----------------------------------------------------------------------------//
// TRAN   TRAN   TRAN   TRAN   TRAN   TRAN   TRAN   TRAN   TRAN   TRAN   TRAN //
// TRAN   TRAN   TRAN   TRAN   TRAN   TRAN   TRAN   TRAN   TRAN   TRAN   TRAN //
//----------------------------------------------------------------------------//
// TIME_VAC_HOLD expired
//----------------------------------------------------------------------------//
// CONDITION   CONDITION   CONDITION   CONDITION   CONDITION   CONDITION   CO //
// CONDITION   CONDITION   CONDITION   CONDITION   CONDITION   CONDITION   CO //
//----------------------------------------------------------------------------//
      A #SQ_TIMER.Q;






  //============================= TRAN FOOTER ==============================//
  // Transition jump control:                                               //
  //------------------------------------------------------------------------//
      A #sqSequencer.STEP.JumpCtrl;
      S #sqSequencer.STEP.Jump;
      S #sqSequencer.STEP.jumpDone[12];

NETWORK
TITLE = S012:t014::TRANS-v: EXIT TRANSITION AND READY THE NEXT STEP
//------------------------------------------------------------------------//
// Check the jump flag and jump to the next step if the transition        //
// condition is true and has set the jump flag:                           //
//------------------------------------------------------------------------//
      A #sqSequencer.STEP.Jump;
      JCN x014;

      R #sqSequencer.STEP.Jump;
      R #sqSequencer.STEP.Finished;

      L 13   ;// Load next STEPNO to jump to if transition satisfied
      T #sqSequencer.STEP.NumberNext;//Next Step13.

      JU COMM            ;// Transition satisfied, Exit, go to next step
x014:      NOP 0;






  //============================= TRAN HEADER ==============================//
  // AUTOCODE   AUTOCODE   AUTOCODE   AUTOCODE   AUTOCODE   AUTOCODE   AUTO //
  // Bypass transition if manual jump:                                      //
  //------------------------------------------------------------------------//
      A #sqSequencer.STEP.Finished;
      A #smc.TRN_AND_JUMP   ;//Manual jump is set Transition as bypassed
      JCN COMM            ;//exit

NETWORK
TITLE = S012::STEP 012:TRAN 015: Pressure above setpoint
//----------------------------------------------------------------------------//
// TRAN   TRAN   TRAN   TRAN   TRAN   TRAN   TRAN   TRAN   TRAN   TRAN   TRAN //
// TRAN   TRAN   TRAN   TRAN   TRAN   TRAN   TRAN   TRAN   TRAN   TRAN   TRAN //
//----------------------------------------------------------------------------//
// Pressure increased above PRES_VAC_FAIL
//----------------------------------------------------------------------------//
// CONDITION   CONDITION   CONDITION   CONDITION   CONDITION   CONDITION   CO //
// CONDITION   CONDITION   CONDITION   CONDITION   CONDITION   CONDITION   CO //
//----------------------------------------------------------------------------//
      O(;
      L #_emc_gas_pi_vessel_pv;
      L #_r_pres_vac_fail;
      >R;
      );






  //============================= TRAN FOOTER ==============================//
  // Transition jump control:                                               //
  //------------------------------------------------------------------------//
      A #sqSequencer.STEP.JumpCtrl;
      S #sqSequencer.STEP.Jump;
      S #sqSequencer.STEP.jumpDone[12];

NETWORK
TITLE = S012:t015::TRANS-v: EXIT TRANSITION AND READY THE NEXT STEP
//------------------------------------------------------------------------//
// Check the jump flag and jump to the next step if the transition        //
// condition is true and has set the jump flag:                           //
//------------------------------------------------------------------------//
      A #sqSequencer.STEP.Jump;
      JCN x015;

      R #sqSequencer.STEP.Jump;
      R #sqSequencer.STEP.Finished;

      L 14   ;// Load next STEPNO to jump to if transition satisfied
      T #sqSequencer.STEP.NumberNext;//Next Step14.

      JU COMM            ;// Transition satisfied, Exit, go to next step
x015:      NOP 0;






  //============================= TRAN HEADER ==============================//
  // AUTOCODE   AUTOCODE   AUTOCODE   AUTOCODE   AUTOCODE   AUTOCODE   AUTO //
  // Bypass transition if manual jump:                                      //
  //------------------------------------------------------------------------//
      A #sqSequencer.STEP.Finished;
      A #smc.TRN_AND_JUMP   ;//Manual jump is set Transition as bypassed
      JCN COMM            ;//exit

NETWORK
TITLE = S012::STEP 012:TRAN 016: Pressure logging timer expired
//----------------------------------------------------------------------------//
// TRAN   TRAN   TRAN   TRAN   TRAN   TRAN   TRAN   TRAN   TRAN   TRAN   TRAN //
// TRAN   TRAN   TRAN   TRAN   TRAN   TRAN   TRAN   TRAN   TRAN   TRAN   TRAN //
//----------------------------------------------------------------------------//
// 30 seconds expired
//----------------------------------------------------------------------------//
// CONDITION   CONDITION   CONDITION   CONDITION   CONDITION   CONDITION   CO //
// CONDITION   CONDITION   CONDITION   CONDITION   CONDITION   CONDITION   CO //
//----------------------------------------------------------------------------//
      A #SQ_TIMER2.Q;






  //============================= TRAN FOOTER ==============================//
  // Transition jump control:                                               //
  //------------------------------------------------------------------------//
      A #sqSequencer.STEP.JumpCtrl;
      S #sqSequencer.STEP.Jump;
      S #sqSequencer.STEP.jumpDone[12];

NETWORK
TITLE = S012:t016::TRANS-v: EXIT TRANSITION AND READY THE NEXT STEP
//------------------------------------------------------------------------//
// Check the jump flag and jump to the next step if the transition        //
// condition is true and has set the jump flag:                           //
//------------------------------------------------------------------------//
      A #sqSequencer.STEP.Jump;
      JCN x016;

      R #sqSequencer.STEP.Jump;
      R #sqSequencer.STEP.Finished;

      L 11   ;// Load next STEPNO to jump to if transition satisfied
      T #sqSequencer.STEP.NumberNext;//Next Step11.

      JU COMM            ;// Transition satisfied, Exit, go to next step
x016:      NOP 0;






NETWORK
TITLE = S012::STEP-012:EXIT TRANSITION:
//========================== STEP TRANSFER ===============================//
// Jump to the common step progression code:                              //
//------------------------------------------------------------------------//
      JU COMM;






NETWORK
TITLE = S013: STEP-13::UO_MX_SETUP : Log actual time vacuum held.
//================================ STEP HEADER ===========================//
// STEP013 STEP013 STEP013 STEP013
// AUTOCODE   AUTOCODE   AUTOCODE   AUTOCODE   AUTOCODE   AUTOCODE   AUTO //
// STEP013 STEP013 STEP013 STEP013
//------------------------------------------------------------------------//
// Log actual time vacuum held.
// Log Mx vessel pressure.
//------------------------------------------------------------------------//
S013:      NOP 0;

      SET;
      R #sqSequencer.STEP.jumpDone[13];
      A #sqSequencer.CMD.Pause;//If paused jump
      JC COMM;

NETWORK
TITLE = S013:STEP-13:Begin Action

      A #sqSequencer.STEP.Finished;
      JC A013;// Exit Action code, Jump to A013 Transition code

    //----------------------------------------------------------------------//
    // Begin step Action:                                                   //
    //----------------------------------------------------------------------//
      A #sqSequencer.STEP.Active;
      JC L013;// Action number loaded, Jump to L013--Step Action List

    //----------------------------------------------------------------------//
    // Load Default/Initial Step action number:                             //
    //----------------------------------------------------------------------//
      S #sqSequencer.STEP.Active;
      S #sqStepTimer.IN;
      L 1;//First Action, Step must contain Minimum one action
      T #sqSequencer.STEP.ActionNumber;

//----------------------------------------------------------------------------//
// Step action list.                                                          //
// aann=mini Action step number(aa) inside main step number(nn)               //
// First Action aa00, Second action ab00, Third ac00, etc.                    //
//----------------------------------------------------------------------------//
L013:      NOP 0;

      L #sqSequencer.STEP.ActionNumber;
      JL r013;//Wrong Action number
      JU _013;//Action error handling
      JU aa13;//ACTION-01


//----------------------------------------------------------------------------//
// More step action in the list can be inserted here, upto ab is tested:      //
//----------------------------------------------------------------------------//
r013:      NOP 0;//Wrong action number
      S #sqSequencer.Error_Fault;
      JU k013;//Exit
_013:      NOP 0;// Action error handling
      JU k013;// Exit






NETWORK
TITLE = S013:: STEP-013:: : ACTION CODE
//================================ ACT HEADER ============================//
// ACTION ACTION ACTION ACTION ACTION ACTION ACTION ACTION ACTION ACTION  //
// AUTOCODE   AUTOCODE   AUTOCODE   AUTOCODE   AUTOCODE   AUTOCODE   AUTO //
// ACTION ACTION ACTION ACTION ACTION ACTION ACTION ACTION ACTION ACTION  //
//------------------------------------------------------------------------//
// //Log actual time vacuum held.
// //Log Mx vessel pressure.
aa13:      NOP 0;

  //------------------------------------------------------------------------//
  // ACT ACT ACT ACT ACT ACT ACT ACT ACT ACT ACT ACT ACT ACT ACT ACT ACT    //
  //------------------------------------------------------------------------//
  //Store Vacuum Hold test end time.
      L "dbCONST".CHRONO.CPU_TIME;
      T #_vacuum_held_end_time;

//Log actual time vacuum held.
      CALL T_DIFF
      {date_type := 'Time_Of_Day', time_type := 'Time'}
      (  IN1                         := #_vacuum_held_end_time ,
         IN2                         := #_vacuum_held_begin_time ,
         OUT                         := #_time_act_vacuum_held
      );
      SET;
      S #_log_time_act_vacuum_held;
      R #sqSeqTimerStart2;

//Log Mx vessel pressure.
      L #_emc_gas_pi_vessel_pv;
      T #_real_pressure_mx;

      SET;
      S #_log_real_pressure_mx;

  //------------------------------------------------------------------------//
  // VERIFY  VERIFY VERIFY VERIFY VERIFY VERIFY VERIFY VERIFY VERIFY VERIFY //
  //------------------------------------------------------------------------//
      A "uncondJump";
      S #sqSequencer.STEP.ActionVerified;//Action verified

  //------------------------------------------------------------------------//
  // Action done:                                                           //
  //------------------------------------------------------------------------//
      O #sqSequencer.STEP.ActionVerified;
      O #smc.NO_VERIFIC     ;//No verification , bypass verification code
      S #sqSequencer.STEP.ActionFinished;






  //============================= STEP FOOTER ==============================//
  // AUTOCODE   AUTOCODE   AUTOCODE   AUTOCODE   AUTOCODE   AUTOCODE   AUTO //
  // Get Ready after action finished:                                       //
  //------------------------------------------------------------------------//
      A #sqSequencer.STEP.ActionFinished;
      JCN k013;

  //------------------------------------------------------------------------//
  // Reset Action finished flag, ready for next step action:                //
  //------------------------------------------------------------------------//
      R #sqSequencer.STEP.ActionVerified;
      R #sqSequencer.STEP.ActionFinished;

  //------------------------------------------------------------------------//
  // If ALL actions are finished:                                           //
  //------------------------------------------------------------------------//
      SET;
      S #sqSequencer.STEP.Finished;
      R #sqSequencer.STEP.Active;
      S #sqSequencer.STEP.Done[13];

  //------------------------------------------------------------------------//
  // End Step action(s):                                                    //
  //------------------------------------------------------------------------//
      JU k013;

//----------------------------------------------------------------------------//
// Finished Step Action(s):                                                   //
//----------------------------------------------------------------------------//
k013:      NOP 0;

      A #sqStepTimerExpired;
      S #sqSequencer.STEP.WithError[13];// Step error flag
      S #sqSequencer.Error_Fault;
      R #sqStepTimer.IN;

NETWORK
TITLE = S013:STEP-013::Begin Transition
//------------------------------------------------------------------------//
// Begin the transition code:                                             //
//------------------------------------------------------------------------//
A013:      NOP 0;
      R #sqStepTimer.IN;






  //============================= TRAN HEADER ==============================//
  // AUTOCODE   AUTOCODE   AUTOCODE   AUTOCODE   AUTOCODE   AUTOCODE   AUTO //
  // Bypass transition if manual jump:                                      //
  //------------------------------------------------------------------------//
      A #sqSequencer.STEP.Finished;
      A #smc.TRN_AND_JUMP   ;//Manual jump is set Transition as bypassed
      JCN COMM            ;//exit

NETWORK
TITLE = S013::STEP 013:TRAN 017: Empty Transition
//----------------------------------------------------------------------------//
// TRAN   TRAN   TRAN   TRAN   TRAN   TRAN   TRAN   TRAN   TRAN   TRAN   TRAN //
// TRAN   TRAN   TRAN   TRAN   TRAN   TRAN   TRAN   TRAN   TRAN   TRAN   TRAN //
//----------------------------------------------------------------------------//
// Empty Transition
//----------------------------------------------------------------------------//
// CONDITION   CONDITION   CONDITION   CONDITION   CONDITION   CONDITION   CO //
// CONDITION   CONDITION   CONDITION   CONDITION   CONDITION   CONDITION   CO //
//----------------------------------------------------------------------------//
      A "uncondJump";






  //============================= TRAN FOOTER ==============================//
  // Transition jump control:                                               //
  //------------------------------------------------------------------------//
      A #sqSequencer.STEP.JumpCtrl;
      S #sqSequencer.STEP.Jump;
      S #sqSequencer.STEP.jumpDone[13];

NETWORK
TITLE = S013:t017::TRANS-v: EXIT TRANSITION AND READY THE NEXT STEP
//------------------------------------------------------------------------//
// Check the jump flag and jump to the next step if the transition        //
// condition is true and has set the jump flag:                           //
//------------------------------------------------------------------------//
      A #sqSequencer.STEP.Jump;
      JCN x017;

      R #sqSequencer.STEP.Jump;
      R #sqSequencer.STEP.Finished;

      L 17   ;// Load next STEPNO to jump to if transition satisfied
      T #sqSequencer.STEP.NumberNext;//Next Step17.

      JU COMM            ;// Transition satisfied, Exit, go to next step
x017:      NOP 0;






NETWORK
TITLE = S013::STEP-013:EXIT TRANSITION:
//========================== STEP TRANSFER ===============================//
// Jump to the common step progression code:                              //
//------------------------------------------------------------------------//
      JU COMM;






NETWORK
TITLE = S014: STEP-14::UO_MX_SETUP : Vacuum Hold failed
//================================ STEP HEADER ===========================//
// STEP014 STEP014 STEP014 STEP014
// AUTOCODE   AUTOCODE   AUTOCODE   AUTOCODE   AUTOCODE   AUTOCODE   AUTO //
// STEP014 STEP014 STEP014 STEP014
//------------------------------------------------------------------------//
// Set flag to raise vacuum failed message and prompt operator.
// Log Mx vessel pressure.
//------------------------------------------------------------------------//
S014:      NOP 0;

      SET;
      R #sqSequencer.STEP.jumpDone[14];
      A #sqSequencer.CMD.Pause;//If paused jump
      JC COMM;

NETWORK
TITLE = S014:STEP-14:Begin Action

      A #sqSequencer.STEP.Finished;
      JC A014;// Exit Action code, Jump to A014 Transition code

    //----------------------------------------------------------------------//
    // Begin step Action:                                                   //
    //----------------------------------------------------------------------//
      A #sqSequencer.STEP.Active;
      JC L014;// Action number loaded, Jump to L014--Step Action List

    //----------------------------------------------------------------------//
    // Load Default/Initial Step action number:                             //
    //----------------------------------------------------------------------//
      S #sqSequencer.STEP.Active;
      S #sqStepTimer.IN;
      L 1;//First Action, Step must contain Minimum one action
      T #sqSequencer.STEP.ActionNumber;

//----------------------------------------------------------------------------//
// Step action list.                                                          //
// aann=mini Action step number(aa) inside main step number(nn)               //
// First Action aa00, Second action ab00, Third ac00, etc.                    //
//----------------------------------------------------------------------------//
L014:      NOP 0;

      L #sqSequencer.STEP.ActionNumber;
      JL r014;//Wrong Action number
      JU _014;//Action error handling
      JU aa14;//ACTION-01


//----------------------------------------------------------------------------//
// More step action in the list can be inserted here, upto ab is tested:      //
//----------------------------------------------------------------------------//
r014:      NOP 0;//Wrong action number
      S #sqSequencer.Error_Fault;
      JU k014;//Exit
_014:      NOP 0;// Action error handling
      JU k014;// Exit






NETWORK
TITLE = S014:: STEP-014:: : ACTION CODE
//================================ ACT HEADER ============================//
// ACTION ACTION ACTION ACTION ACTION ACTION ACTION ACTION ACTION ACTION  //
// AUTOCODE   AUTOCODE   AUTOCODE   AUTOCODE   AUTOCODE   AUTOCODE   AUTO //
// ACTION ACTION ACTION ACTION ACTION ACTION ACTION ACTION ACTION ACTION  //
//------------------------------------------------------------------------//
// //Set flag to raise vacuum failed message and prompt operator.
// //Log Mx vessel pressure.
aa14:      NOP 0;

  //------------------------------------------------------------------------//
  // ACT ACT ACT ACT ACT ACT ACT ACT ACT ACT ACT ACT ACT ACT ACT ACT ACT    //
  //------------------------------------------------------------------------//
  //Set flag to raise vacuum failed message and prompt operator.
      SET;
      S #_log_real_not_held;
      S #_prompt_not_held;


// Stop timer
      SET;
      R #sqSeqTimerStart;
      R #sqSeqTimerStart2;

//Log Mx vessel pressure.
      L #_emc_gas_pi_vessel_pv;
      T #_real_not_held;

  //------------------------------------------------------------------------//
  // VERIFY  VERIFY VERIFY VERIFY VERIFY VERIFY VERIFY VERIFY VERIFY VERIFY //
  //------------------------------------------------------------------------//
      A "uncondJump";
      S #sqSequencer.STEP.ActionVerified;//Action verified

  //------------------------------------------------------------------------//
  // Action done:                                                           //
  //------------------------------------------------------------------------//
      O #sqSequencer.STEP.ActionVerified;
      O #smc.NO_VERIFIC     ;//No verification , bypass verification code
      S #sqSequencer.STEP.ActionFinished;






  //============================= STEP FOOTER ==============================//
  // AUTOCODE   AUTOCODE   AUTOCODE   AUTOCODE   AUTOCODE   AUTOCODE   AUTO //
  // Get Ready after action finished:                                       //
  //------------------------------------------------------------------------//
      A #sqSequencer.STEP.ActionFinished;
      JCN k014;

  //------------------------------------------------------------------------//
  // Reset Action finished flag, ready for next step action:                //
  //------------------------------------------------------------------------//
      R #sqSequencer.STEP.ActionVerified;
      R #sqSequencer.STEP.ActionFinished;

  //------------------------------------------------------------------------//
  // If ALL actions are finished:                                           //
  //------------------------------------------------------------------------//
      SET;
      S #sqSequencer.STEP.Finished;
      R #sqSequencer.STEP.Active;
      S #sqSequencer.STEP.Done[14];

  //------------------------------------------------------------------------//
  // End Step action(s):                                                    //
  //------------------------------------------------------------------------//
      JU k014;

//----------------------------------------------------------------------------//
// Finished Step Action(s):                                                   //
//----------------------------------------------------------------------------//
k014:      NOP 0;

      A #sqStepTimerExpired;
      S #sqSequencer.STEP.WithError[14];// Step error flag
      S #sqSequencer.Error_Fault;
      R #sqStepTimer.IN;

NETWORK
TITLE = S014:STEP-014::Begin Transition
//------------------------------------------------------------------------//
// Begin the transition code:                                             //
//------------------------------------------------------------------------//
A014:      NOP 0;
      R #sqStepTimer.IN;






  //============================= TRAN HEADER ==============================//
  // AUTOCODE   AUTOCODE   AUTOCODE   AUTOCODE   AUTOCODE   AUTOCODE   AUTO //
  // Bypass transition if manual jump:                                      //
  //------------------------------------------------------------------------//
      A #sqSequencer.STEP.Finished;
      A #smc.TRN_AND_JUMP   ;//Manual jump is set Transition as bypassed
      JCN COMM            ;//exit

NETWORK
TITLE = S014::STEP 014:TRAN 018: No try?
//----------------------------------------------------------------------------//
// TRAN   TRAN   TRAN   TRAN   TRAN   TRAN   TRAN   TRAN   TRAN   TRAN   TRAN //
// TRAN   TRAN   TRAN   TRAN   TRAN   TRAN   TRAN   TRAN   TRAN   TRAN   TRAN //
//----------------------------------------------------------------------------//
// Operator don't want to try again.
//----------------------------------------------------------------------------//
// CONDITION   CONDITION   CONDITION   CONDITION   CONDITION   CONDITION   CO //
// CONDITION   CONDITION   CONDITION   CONDITION   CONDITION   CONDITION   CO //
//----------------------------------------------------------------------------//
      A #_prompt_not_held_confirm_no;






  //============================= TRAN FOOTER ==============================//
  // Transition jump control:                                               //
  //------------------------------------------------------------------------//
      A #sqSequencer.STEP.JumpCtrl;
      S #sqSequencer.STEP.Jump;
      S #sqSequencer.STEP.jumpDone[14];

NETWORK
TITLE = S014:t018::TRANS-v: EXIT TRANSITION AND READY THE NEXT STEP
//------------------------------------------------------------------------//
// Check the jump flag and jump to the next step if the transition        //
// condition is true and has set the jump flag:                           //
//------------------------------------------------------------------------//
      A #sqSequencer.STEP.Jump;
      JCN x018;

      R #sqSequencer.STEP.Jump;
      R #sqSequencer.STEP.Finished;

      L 15   ;// Load next STEPNO to jump to if transition satisfied
      T #sqSequencer.STEP.NumberNext;//Next Step15.

      JU COMM            ;// Transition satisfied, Exit, go to next step
x018:      NOP 0;






  //============================= TRAN HEADER ==============================//
  // AUTOCODE   AUTOCODE   AUTOCODE   AUTOCODE   AUTOCODE   AUTOCODE   AUTO //
  // Bypass transition if manual jump:                                      //
  //------------------------------------------------------------------------//
      A #sqSequencer.STEP.Finished;
      A #smc.TRN_AND_JUMP   ;//Manual jump is set Transition as bypassed
      JCN COMM            ;//exit

NETWORK
TITLE = S014::STEP 014:TRAN 019: Try again?
//----------------------------------------------------------------------------//
// TRAN   TRAN   TRAN   TRAN   TRAN   TRAN   TRAN   TRAN   TRAN   TRAN   TRAN //
// TRAN   TRAN   TRAN   TRAN   TRAN   TRAN   TRAN   TRAN   TRAN   TRAN   TRAN //
//----------------------------------------------------------------------------//
// Operator want to try again.
//----------------------------------------------------------------------------//
// CONDITION   CONDITION   CONDITION   CONDITION   CONDITION   CONDITION   CO //
// CONDITION   CONDITION   CONDITION   CONDITION   CONDITION   CONDITION   CO //
//----------------------------------------------------------------------------//
      A #_prompt_not_held_confirm_yes;






  //============================= TRAN FOOTER ==============================//
  // Transition jump control:                                               //
  //------------------------------------------------------------------------//
      A #sqSequencer.STEP.JumpCtrl;
      S #sqSequencer.STEP.Jump;
      S #sqSequencer.STEP.jumpDone[14];

NETWORK
TITLE = S014:t019::TRANS-v: EXIT TRANSITION AND READY THE NEXT STEP
//------------------------------------------------------------------------//
// Check the jump flag and jump to the next step if the transition        //
// condition is true and has set the jump flag:                           //
//------------------------------------------------------------------------//
      A #sqSequencer.STEP.Jump;
      JCN x019;

      R #sqSequencer.STEP.Jump;
      R #sqSequencer.STEP.Finished;

      L 16   ;// Load next STEPNO to jump to if transition satisfied
      T #sqSequencer.STEP.NumberNext;//Next Step16.

      JU COMM            ;// Transition satisfied, Exit, go to next step
x019:      NOP 0;






NETWORK
TITLE = S014::STEP-014:EXIT TRANSITION:
//========================== STEP TRANSFER ===============================//
// Jump to the common step progression code:                              //
//------------------------------------------------------------------------//
      JU COMM;






NETWORK
TITLE = S015: STEP-15::UO_MX_SETUP : Log operator abort
//================================ STEP HEADER ===========================//
// STEP015 STEP015 STEP015 STEP015
// AUTOCODE   AUTOCODE   AUTOCODE   AUTOCODE   AUTOCODE   AUTOCODE   AUTO //
// STEP015 STEP015 STEP015 STEP015
//------------------------------------------------------------------------//
// Log operator abort.
//------------------------------------------------------------------------//
S015:      NOP 0;

      SET;
      R #sqSequencer.STEP.jumpDone[15];
      A #sqSequencer.CMD.Pause;//If paused jump
      JC COMM;

NETWORK
TITLE = S015:STEP-15:Begin Action

      A #sqSequencer.STEP.Finished;
      JC A015;// Exit Action code, Jump to A015 Transition code

    //----------------------------------------------------------------------//
    // Begin step Action:                                                   //
    //----------------------------------------------------------------------//
      A #sqSequencer.STEP.Active;
      JC L015;// Action number loaded, Jump to L015--Step Action List

    //----------------------------------------------------------------------//
    // Load Default/Initial Step action number:                             //
    //----------------------------------------------------------------------//
      S #sqSequencer.STEP.Active;
      S #sqStepTimer.IN;
      L 1;//First Action, Step must contain Minimum one action
      T #sqSequencer.STEP.ActionNumber;

//----------------------------------------------------------------------------//
// Step action list.                                                          //
// aann=mini Action step number(aa) inside main step number(nn)               //
// First Action aa00, Second action ab00, Third ac00, etc.                    //
//----------------------------------------------------------------------------//
L015:      NOP 0;

      L #sqSequencer.STEP.ActionNumber;
      JL r015;//Wrong Action number
      JU _015;//Action error handling
      JU aa15;//ACTION-01


//----------------------------------------------------------------------------//
// More step action in the list can be inserted here, upto ab is tested:      //
//----------------------------------------------------------------------------//
r015:      NOP 0;//Wrong action number
      S #sqSequencer.Error_Fault;
      JU k015;//Exit
_015:      NOP 0;// Action error handling
      JU k015;// Exit






NETWORK
TITLE = S015:: STEP-015:: : ACTION CODE
//================================ ACT HEADER ============================//
// ACTION ACTION ACTION ACTION ACTION ACTION ACTION ACTION ACTION ACTION  //
// AUTOCODE   AUTOCODE   AUTOCODE   AUTOCODE   AUTOCODE   AUTOCODE   AUTO //
// ACTION ACTION ACTION ACTION ACTION ACTION ACTION ACTION ACTION ACTION  //
//------------------------------------------------------------------------//
// //Log operator abort.
aa15:      NOP 0;

  //------------------------------------------------------------------------//
  // ACT ACT ACT ACT ACT ACT ACT ACT ACT ACT ACT ACT ACT ACT ACT ACT ACT    //
  //------------------------------------------------------------------------//
  //Log operator abort.
      SET;
      S #_log_msg_not_held_abort;
      R #_prompt_not_held_confirm_no;

  //------------------------------------------------------------------------//
  // VERIFY  VERIFY VERIFY VERIFY VERIFY VERIFY VERIFY VERIFY VERIFY VERIFY //
  //------------------------------------------------------------------------//
      A "uncondJump";
      S #sqSequencer.STEP.ActionVerified;//Action verified

  //------------------------------------------------------------------------//
  // Action done:                                                           //
  //------------------------------------------------------------------------//
      O #sqSequencer.STEP.ActionVerified;
      O #smc.NO_VERIFIC     ;//No verification , bypass verification code
      S #sqSequencer.STEP.ActionFinished;






  //============================= STEP FOOTER ==============================//
  // AUTOCODE   AUTOCODE   AUTOCODE   AUTOCODE   AUTOCODE   AUTOCODE   AUTO //
  // Get Ready after action finished:                                       //
  //------------------------------------------------------------------------//
      A #sqSequencer.STEP.ActionFinished;
      JCN k015;

  //------------------------------------------------------------------------//
  // Reset Action finished flag, ready for next step action:                //
  //------------------------------------------------------------------------//
      R #sqSequencer.STEP.ActionVerified;
      R #sqSequencer.STEP.ActionFinished;

  //------------------------------------------------------------------------//
  // If ALL actions are finished:                                           //
  //------------------------------------------------------------------------//
      SET;
      S #sqSequencer.STEP.Finished;
      R #sqSequencer.STEP.Active;
      S #sqSequencer.STEP.Done[15];

  //------------------------------------------------------------------------//
  // End Step action(s):                                                    //
  //------------------------------------------------------------------------//
      JU k015;

//----------------------------------------------------------------------------//
// Finished Step Action(s):                                                   //
//----------------------------------------------------------------------------//
k015:      NOP 0;

      A #sqStepTimerExpired;
      S #sqSequencer.STEP.WithError[15];// Step error flag
      S #sqSequencer.Error_Fault;
      R #sqStepTimer.IN;

NETWORK
TITLE = S015:STEP-015::Begin Transition
//------------------------------------------------------------------------//
// Begin the transition code:                                             //
//------------------------------------------------------------------------//
A015:      NOP 0;
      R #sqStepTimer.IN;






  //============================= TRAN HEADER ==============================//
  // AUTOCODE   AUTOCODE   AUTOCODE   AUTOCODE   AUTOCODE   AUTOCODE   AUTO //
  // Bypass transition if manual jump:                                      //
  //------------------------------------------------------------------------//
      A #sqSequencer.STEP.Finished;
      A #smc.TRN_AND_JUMP   ;//Manual jump is set Transition as bypassed
      JCN COMM            ;//exit

NETWORK
TITLE = S015::STEP 015:TRAN 020: Empty Transition
//----------------------------------------------------------------------------//
// TRAN   TRAN   TRAN   TRAN   TRAN   TRAN   TRAN   TRAN   TRAN   TRAN   TRAN //
// TRAN   TRAN   TRAN   TRAN   TRAN   TRAN   TRAN   TRAN   TRAN   TRAN   TRAN //
//----------------------------------------------------------------------------//
// Empty Transition
//----------------------------------------------------------------------------//
// CONDITION   CONDITION   CONDITION   CONDITION   CONDITION   CONDITION   CO //
// CONDITION   CONDITION   CONDITION   CONDITION   CONDITION   CONDITION   CO //
//----------------------------------------------------------------------------//
      A "uncondJump";






  //============================= TRAN FOOTER ==============================//
  // Transition jump control:                                               //
  //------------------------------------------------------------------------//
      A #sqSequencer.STEP.JumpCtrl;
      S #sqSequencer.STEP.Jump;
      S #sqSequencer.STEP.jumpDone[15];

NETWORK
TITLE = S015:t020::TRANS-v: EXIT TRANSITION AND READY THE NEXT STEP
//------------------------------------------------------------------------//
// Check the jump flag and jump to the next step if the transition        //
// condition is true and has set the jump flag:                           //
//------------------------------------------------------------------------//
      A #sqSequencer.STEP.Jump;
      JCN x020;

      R #sqSequencer.STEP.Jump;
      R #sqSequencer.STEP.Finished;

      L 17   ;// Load next STEPNO to jump to if transition satisfied
      T #sqSequencer.STEP.NumberNext;//Next Step17.

      JU COMM            ;// Transition satisfied, Exit, go to next step
x020:      NOP 0;






NETWORK
TITLE = S015::STEP-015:EXIT TRANSITION:
//========================== STEP TRANSFER ===============================//
// Jump to the common step progression code:                              //
//------------------------------------------------------------------------//
      JU COMM;






NETWORK
TITLE = S016: STEP-16::UO_MX_SETUP : Log operator repeat
//================================ STEP HEADER ===========================//
// STEP016 STEP016 STEP016 STEP016
// AUTOCODE   AUTOCODE   AUTOCODE   AUTOCODE   AUTOCODE   AUTOCODE   AUTO //
// STEP016 STEP016 STEP016 STEP016
//------------------------------------------------------------------------//
// Log operator repeat
//------------------------------------------------------------------------//
S016:      NOP 0;

      SET;
      R #sqSequencer.STEP.jumpDone[16];
      A #sqSequencer.CMD.Pause;//If paused jump
      JC COMM;

NETWORK
TITLE = S016:STEP-16:Begin Action

      A #sqSequencer.STEP.Finished;
      JC A016;// Exit Action code, Jump to A016 Transition code

    //----------------------------------------------------------------------//
    // Begin step Action:                                                   //
    //----------------------------------------------------------------------//
      A #sqSequencer.STEP.Active;
      JC L016;// Action number loaded, Jump to L016--Step Action List

    //----------------------------------------------------------------------//
    // Load Default/Initial Step action number:                             //
    //----------------------------------------------------------------------//
      S #sqSequencer.STEP.Active;
      S #sqStepTimer.IN;
      L 1;//First Action, Step must contain Minimum one action
      T #sqSequencer.STEP.ActionNumber;

//----------------------------------------------------------------------------//
// Step action list.                                                          //
// aann=mini Action step number(aa) inside main step number(nn)               //
// First Action aa00, Second action ab00, Third ac00, etc.                    //
//----------------------------------------------------------------------------//
L016:      NOP 0;

      L #sqSequencer.STEP.ActionNumber;
      JL r016;//Wrong Action number
      JU _016;//Action error handling
      JU aa16;//ACTION-01


//----------------------------------------------------------------------------//
// More step action in the list can be inserted here, upto ab is tested:      //
//----------------------------------------------------------------------------//
r016:      NOP 0;//Wrong action number
      S #sqSequencer.Error_Fault;
      JU k016;//Exit
_016:      NOP 0;// Action error handling
      JU k016;// Exit






NETWORK
TITLE = S016:: STEP-016:: : ACTION CODE
//================================ ACT HEADER ============================//
// ACTION ACTION ACTION ACTION ACTION ACTION ACTION ACTION ACTION ACTION  //
// AUTOCODE   AUTOCODE   AUTOCODE   AUTOCODE   AUTOCODE   AUTOCODE   AUTO //
// ACTION ACTION ACTION ACTION ACTION ACTION ACTION ACTION ACTION ACTION  //
//------------------------------------------------------------------------//
// //Log operator repeat
aa16:      NOP 0;

  //------------------------------------------------------------------------//
  // ACT ACT ACT ACT ACT ACT ACT ACT ACT ACT ACT ACT ACT ACT ACT ACT ACT    //
  //------------------------------------------------------------------------//
  //Log operator repeat.
      SET;
      S #_log_msg_not_held_repeat;
      R #_prompt_not_held_confirm_yes;

  //------------------------------------------------------------------------//
  // VERIFY  VERIFY VERIFY VERIFY VERIFY VERIFY VERIFY VERIFY VERIFY VERIFY //
  //------------------------------------------------------------------------//
      A "uncondJump";
      S #sqSequencer.STEP.ActionVerified;//Action verified

  //------------------------------------------------------------------------//
  // Action done:                                                           //
  //------------------------------------------------------------------------//
      O #sqSequencer.STEP.ActionVerified;
      O #smc.NO_VERIFIC     ;//No verification , bypass verification code
      S #sqSequencer.STEP.ActionFinished;






  //============================= STEP FOOTER ==============================//
  // AUTOCODE   AUTOCODE   AUTOCODE   AUTOCODE   AUTOCODE   AUTOCODE   AUTO //
  // Get Ready after action finished:                                       //
  //------------------------------------------------------------------------//
      A #sqSequencer.STEP.ActionFinished;
      JCN k016;

  //------------------------------------------------------------------------//
  // Reset Action finished flag, ready for next step action:                //
  //------------------------------------------------------------------------//
      R #sqSequencer.STEP.ActionVerified;
      R #sqSequencer.STEP.ActionFinished;

  //------------------------------------------------------------------------//
  // If ALL actions are finished:                                           //
  //------------------------------------------------------------------------//
      SET;
      S #sqSequencer.STEP.Finished;
      R #sqSequencer.STEP.Active;
      S #sqSequencer.STEP.Done[16];

  //------------------------------------------------------------------------//
  // End Step action(s):                                                    //
  //------------------------------------------------------------------------//
      JU k016;

//----------------------------------------------------------------------------//
// Finished Step Action(s):                                                   //
//----------------------------------------------------------------------------//
k016:      NOP 0;

      A #sqStepTimerExpired;
      S #sqSequencer.STEP.WithError[16];// Step error flag
      S #sqSequencer.Error_Fault;
      R #sqStepTimer.IN;

NETWORK
TITLE = S016:STEP-016::Begin Transition
//------------------------------------------------------------------------//
// Begin the transition code:                                             //
//------------------------------------------------------------------------//
A016:      NOP 0;
      R #sqStepTimer.IN;






